// TIA Portal V19 export
TYPE "UDT_Word"
   STRUCT
      b_0 : Bool := false;
      b_1 : Bool := false;
      b_2 : Bool := false;
      b_3 : Bool := false;
      b_4 : Bool := false;
      b_5 : Bool := false;
      b_6 : Bool := false;
      b_7 : Bool := false;
      b_8 : Bool := false;
      b_9 : Bool := false;
      b_10 : Bool := false;
      b_11 : Bool := false;
      b_12 : Bool := false;
      b_13 : Bool := false;
      b_14 : Bool := false;
      b_15 : Bool := false;
   END_STRUCT;
END_TYPE
